// TIA Portal V21 export
FUNCTION_BLOCK "FB301"   // FB301, LAD
TITLE = FB301
{ S7_Optimized_Access := 'TRUE' }
AUTHOR : PRECISE
FAMILY : PRECISE
// FILLING/FINAL VOLUME MAKEUP
// stored: AutoNumber false, MemoryReserve 100, SetENOAutomatically false
   VAR_INPUT
      Enable : Bool;
      Disable : Bool;
      Fault : Bool;
      SecPulse : Bool;
      AlwaysTrue : Bool;
      StartConfirmationPopupSel : Bool;   // StartConfirmationPopupSel: 0-NO/1-YES
      EndConfirmationPopupSel : Bool;   // EndConfirmationPopupSel: 0-NO/1-YES
      FillModeSel : Int;   // Filling Mode Selection: 0-Auto/1-Manual
      FillMethodSel : Int;   // Filling Method Selection: 0-Weight/1-Time
      FillTimeBaseSel : Bool;   // Filling Time Base Selection: 0-second/1-minute
      FillLineSel : Int;   // Filling Line Selection: 0-J tube/1-SBI
      InitialDrainSel : Bool;
      SBIPulsingSel : Bool;
      FinalVolumeMakeupSel : Bool;
      PurgingSel : Bool;
      UtilitySel : Bool;   // Utility Selection: 0-PW/1-WFI
      FillQuantity : Real := 10.0;   // For Filling Method Slection: 0-Weight
      FillTimeMin : Int := 1;   // For Filling Method Slection: 1-Time
      FillTimeSec : Int := 30;   // For Filling Method Slection: 1-Time
      ActualQuantity : Real;   // For Filling Method Slection: 0-Weight
      InflightQuantity : Real;   // For Filling Method Slection: 0-Weight
      ZDVDelay : Int := 3;
      InitialDrainDelay : Int := 10;   // For Initial Drain Selection: Yes
      PurgingTime : Int := 10;   // For Purging Selection: Yes
      SBIOnTime : Int := 3;   // For SBI Pulsing Selection: Yes
      SBIOffTime : Int := 4;   // For SBI Pulsing Selection: Yes
      SetQuantitytoStartPulsing : Real := 10.0;   // For SBI Pulsing Selection: Yes
      FillQuantityTolerance : Real := 3.0;   // For Filling Method Slection: 0-Weight
      PrintInetrval : Int;
   END_VAR
   VAR_OUTPUT
      PWZDV : Bool;   // For Utility Selection: 0-PW
      WFIZDV : Bool;   // For Utility Selection: 1-WFI
      PWLineValves : Bool;   // For Utility Selection: 0-PW
      WFILineValves : Bool;   // For Utility Selection: 1-WFI
      InitialDrainValves : Bool;   // For Initial Drain Selection: Yes
      SBIValve : Bool;   // For Filling Line Selection: 1-SBI
      JTubeValve : Bool;   // For Filling Line Selection: 0-J tube
      AirInletValve : Bool;   // For Purging Selection: Yes
      StartConfirmationPopup : Bool;   // For Start Confirmation Popup Selection: Yes
      EndConfirmationPopup : Bool;   // For End Confirmation Popup Selection: Yes
      ManualPopup : Bool;   // For Filling Mode Selection: 1-Manual
      AlarmFillQuantityExeeded : Bool;
      FillTimeMinPV : DInt;   // For Filling Method Slection: 1-Time
      FillTimeSecPV : DInt;   // For Filling Method Slection: 1-Time
      PrintTrigger : Bool;
      PrintWord : Int;
      PrintStatus : String[50];
   END_VAR
   VAR_IN_OUT
      Start : Bool;
      Stop : Bool;
      Reset : Bool;
      StartConfirmationAck : Bool;   // For Start Confirmation Popup Selection: Yes
      EndConfirmationAck : Bool;   // For End Confirmation Popup Selection: Yes
      ManualAck : Bool;   // For Filling Mode Selection: 1-Manual
      AlarmAck : Bool;
      SpareBtn1 : Bool;
      Running : Bool;
      Selected : Bool;
      Paused : Bool;
      StartConfirmationPopupTemp : Bool;   // For Start Confirmation Popup Selection: Yes
      EndConfirmationPopupTemp : Bool;   // For End Confirmation Popup Selection: Yes
      ManualPopupTemp : Bool;   // For Filling Mode Selection: 1-Manual
      InitialDrainDelayStarted : Bool;
      InitialDrainDelayOver : Bool;
      FillStarted : Bool;
      FillOver : Bool;
      FillOverTemp : Bool;
      InitialDrainDelayPV : Int;
      ActualFillQuantityCalc : Real;   // For Filling Method Slection: 0-Weight
      ActualFillQuantity : Real;   // For Filling Method Slection: 0-Weight
      PulsingStartWeight : Real;   // For SBI Pulsing Selection: Yes
      PurgingTimePV : Int;   // For Purging Selection: Yes
      FillQuantityToleranceCalc : Real := 3.0;   // For Filling Method Slection: 0-Weight
      VesselMaxWeight : Real := 1000.0;
      ResetBatchTimer : Bool;
   END_VAR
   VAR
      ValveOnDelayPV : Int;
      ValveOffDelayPV : Int;
      PrintTriggerTemp : Bool;
      RE1 : Bool;
      RE2 : Bool;
      RE3 : Bool;
      RE4 : Bool;
      RE5 : Bool;
      RE6 : Bool;
      RE7 : Bool;
      FillTimer { S7_SetPoint := 'True'} : "FB101";
      SBIPulsing { S7_SetPoint := 'True'} : "FB102";
      PrintTriggerResetTimer { S7_SetPoint := 'True'} : TON_TIME;
      BtnResetTimer { S7_SetPoint := 'True'} : TON_TIME;
      IEC_Counter_0_Instance { S7_SetPoint := 'True'} : CTU_INT;
   END_VAR
   VAR_TEMP
      STATUS1 : String[40];
      STATUS2 : String[40];
      STATUS3 : String[40];
      STATUS4 : String[40];
      STATUS5 : String[40];
   END_VAR
   VAR_TEMP   // added for the SCL form of the ladder/FBD networks
      _w1 : Bool;
      _w2 : Bool;
      _w3 : Bool;
      _w4 : Bool;
      _w5 : Bool;
      _w6 : Bool;
   END_VAR
BEGIN

REGION Network 1: Running
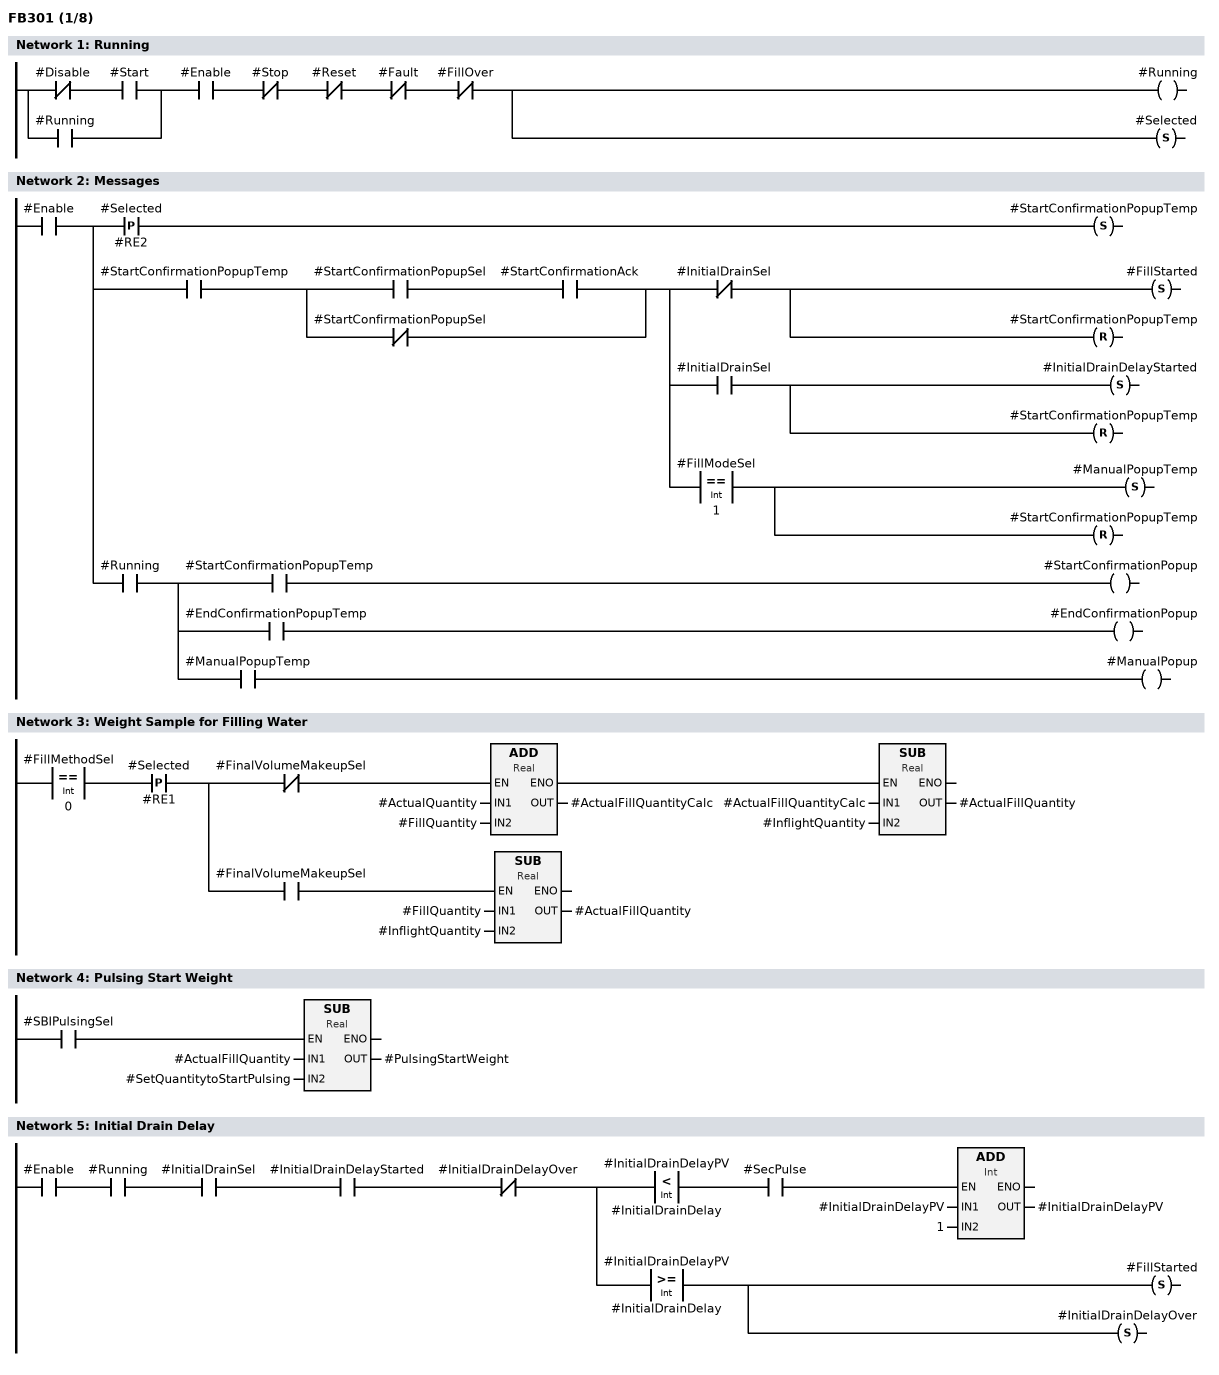
   RUNG wire#powerrail
      I_Contact( #Disable )
      Contact( #Start )
      wire#w1
      Contact( #Enable )
      I_Contact( #Stop )
      I_Contact( #Reset )
      I_Contact( #Fault )
      I_Contact( #FillOver )
      wire#w2
      Coil( #Running )
   END_RUNG
   RUNG wire#powerrail
      Contact( #Running )
   END_RUNG wire#w1
   RUNG wire#w2
      S_Coil( #Selected )
   END_RUNG
   // the same network as SCL:
   #Running := ((NOT #Disable AND #Start) OR #Running) AND #Enable AND NOT #Stop AND NOT #Reset AND NOT #Fault AND NOT #FillOver;
   IF #Running THEN #Selected := TRUE; END_IF;
END_REGION

REGION Network 2: Messages
   RUNG wire#powerrail
      Contact( #Enable )
      wire#w1
      P_Contact(operand := #Selected, bit := #RE2)
      S_Coil( #StartConfirmationPopupTemp )
   END_RUNG
   RUNG wire#w1
      Contact( #StartConfirmationPopupTemp )
      wire#w2
      Contact( #StartConfirmationPopupSel )
      Contact( #StartConfirmationAck )
      wire#w3
      I_Contact( #InitialDrainSel )
      wire#w4
      S_Coil( #FillStarted )
   END_RUNG
   RUNG wire#w2
      I_Contact( #StartConfirmationPopupSel )
   END_RUNG wire#w3
   RUNG wire#w4
      R_Coil( #StartConfirmationPopupTemp )
   END_RUNG
   RUNG wire#w3
      Contact( #InitialDrainSel )
      wire#w5
      S_Coil( #InitialDrainDelayStarted )
   END_RUNG
   RUNG wire#w5
      R_Coil( #StartConfirmationPopupTemp )
   END_RUNG
   RUNG wire#w3
      { S7_Templates := "SrcType := Int" } EQ_Contact(in1 := #FillModeSel, in2 := 1)
      wire#w6
      S_Coil( #ManualPopupTemp )
   END_RUNG
   RUNG wire#w6
      R_Coil( #StartConfirmationPopupTemp )
   END_RUNG
   RUNG wire#w1
      Contact( #Running )
      wire#w7
      Contact( #StartConfirmationPopupTemp )
      Coil( #StartConfirmationPopup )
   END_RUNG
   RUNG wire#w7
      Contact( #EndConfirmationPopupTemp )
      Coil( #EndConfirmationPopup )
   END_RUNG
   RUNG wire#w7
      Contact( #ManualPopupTemp )
      Coil( #ManualPopup )
   END_RUNG
   // the same network as SCL:
   #_w1 := #Enable AND #Selected AND NOT #RE2;   // rising edge of #Selected
   #RE2 := #Selected;
   IF #_w1 THEN #StartConfirmationPopupTemp := TRUE; END_IF;
   #_w2 := #Enable AND #StartConfirmationPopupTemp AND ((#StartConfirmationPopupSel AND #StartConfirmationAck) OR NOT #StartConfirmationPopupSel);
   IF #_w2 AND NOT #InitialDrainSel THEN
       #FillStarted := TRUE;
       #StartConfirmationPopupTemp := FALSE;
   END_IF;
   IF #_w2 AND #InitialDrainSel THEN
       #InitialDrainDelayStarted := TRUE;
       #StartConfirmationPopupTemp := FALSE;
   END_IF;
   IF #_w2 AND (#FillModeSel = 1) THEN
       #ManualPopupTemp := TRUE;
       #StartConfirmationPopupTemp := FALSE;
   END_IF;
   #_w3 := #Enable AND #Running;
   #StartConfirmationPopup := #_w3 AND #StartConfirmationPopupTemp;
   #EndConfirmationPopup := #_w3 AND #EndConfirmationPopupTemp;
   #ManualPopup := #_w3 AND #ManualPopupTemp;
END_REGION

REGION Network 3: Weight Sample for Filling Water
   RUNG wire#powerrail
      { S7_Templates := "SrcType := Int" } EQ_Contact(in1 := #FillMethodSel, in2 := 0)
      P_Contact(operand := #Selected, bit := #RE1)
      wire#w1
      I_Contact( #FinalVolumeMakeupSel )
      { S7_Templates := "SrcType := Real"; S7_GenerateENO := "TRUE" } Add(in1 := #ActualQuantity, in2 := #FillQuantity, out => #ActualFillQuantityCalc)
      { S7_Templates := "SrcType := Real"; S7_GenerateENO := "TRUE" } Sub(in1 := #ActualFillQuantityCalc, in2 := #InflightQuantity, out => #ActualFillQuantity)
   END_RUNG
   RUNG wire#w1
      Contact( #FinalVolumeMakeupSel )
      { S7_Templates := "SrcType := Real"; S7_GenerateENO := "TRUE" } Sub(in1 := #FillQuantity, in2 := #InflightQuantity, out => #ActualFillQuantity)
   END_RUNG
   // the same network as SCL:
   // ENO of a box is taken as its EN; it also drops when the box reports an error
   #_w1 := (#FillMethodSel = 0) AND #Selected AND NOT #RE1;   // rising edge of #Selected
   #RE1 := #Selected;
   IF #_w1 AND NOT #FinalVolumeMakeupSel THEN
       #ActualFillQuantityCalc := #ActualQuantity + #FillQuantity;
       #ActualFillQuantity := #ActualFillQuantityCalc - #InflightQuantity;
   END_IF;
   IF #_w1 AND #FinalVolumeMakeupSel THEN #ActualFillQuantity := #FillQuantity - #InflightQuantity; END_IF;
END_REGION

REGION Network 4: Pulsing Start Weight
   RUNG wire#powerrail
      Contact( #SBIPulsingSel )
      { S7_Templates := "SrcType := Real"; S7_GenerateENO := "TRUE" } Sub(in1 := #ActualFillQuantity, in2 := #SetQuantitytoStartPulsing, out => #PulsingStartWeight)
   END_RUNG
   // the same network as SCL:
   IF #SBIPulsingSel THEN #PulsingStartWeight := #ActualFillQuantity - #SetQuantitytoStartPulsing; END_IF;
END_REGION

REGION Network 5: Initial Drain Delay
   RUNG wire#powerrail
      Contact( #Enable )
      Contact( #Running )
      Contact( #InitialDrainSel )
      Contact( #InitialDrainDelayStarted )
      I_Contact( #InitialDrainDelayOver )
      wire#w1
      { S7_Templates := "SrcType := Int" } LT_Contact(in1 := #InitialDrainDelayPV, in2 := #InitialDrainDelay)
      Contact( #SecPulse )
      { S7_Templates := "SrcType := Int"; S7_GenerateENO := "TRUE" } Add(in1 := #InitialDrainDelayPV, in2 := 1, out => #InitialDrainDelayPV)
   END_RUNG
   RUNG wire#w1
      { S7_Templates := "SrcType := Int" } GE_Contact(in1 := #InitialDrainDelayPV, in2 := #InitialDrainDelay)
      wire#w2
      S_Coil( #FillStarted )
   END_RUNG
   RUNG wire#w2
      S_Coil( #InitialDrainDelayOver )
   END_RUNG
   // the same network as SCL:
   #_w1 := #Enable AND #Running AND #InitialDrainSel AND #InitialDrainDelayStarted AND NOT #InitialDrainDelayOver;
   IF #_w1 AND (#InitialDrainDelayPV < #InitialDrainDelay) AND #SecPulse THEN
       #InitialDrainDelayPV := #InitialDrainDelayPV + 1;
   END_IF;
   IF #_w1 AND (#InitialDrainDelayPV >= #InitialDrainDelay) THEN
       #FillStarted := TRUE;
       #InitialDrainDelayOver := TRUE;
   END_IF;
END_REGION

REGION Network 6: Fill Timer
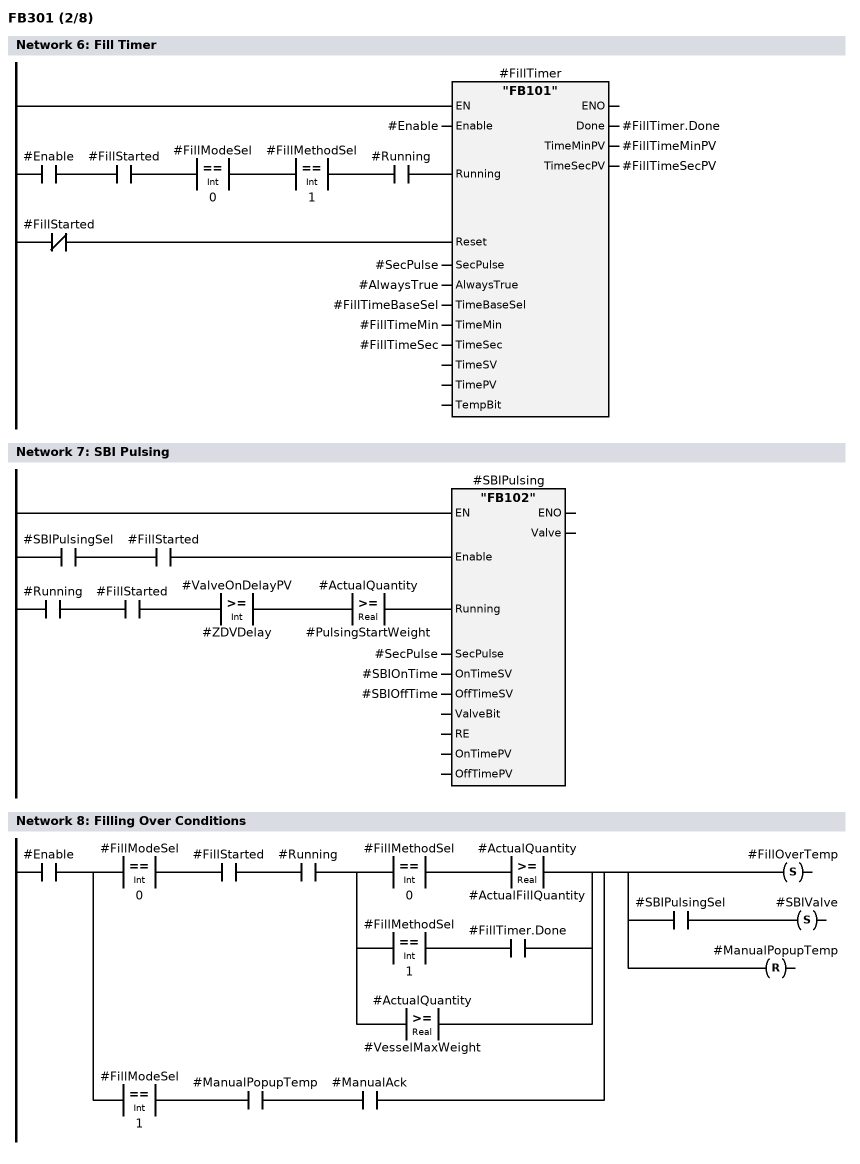
   RUNG wire#powerrail
      #FillTimer(Running := wire#w1, Reset := wire#w2, Enable := #Enable, SecPulse := #SecPulse, AlwaysTrue := #AlwaysTrue, TimeBaseSel := #FillTimeBaseSel, TimeMin := #FillTimeMin, TimeSec := #FillTimeSec, TimeSV :=, TimePV :=, TempBit :=, Done => #FillTimer.Done, TimeMinPV => #FillTimeMinPV, TimeSecPV => #FillTimeSecPV)
   END_RUNG
   RUNG wire#powerrail
      Contact( #Enable )
      Contact( #FillStarted )
      { S7_Templates := "SrcType := Int" } EQ_Contact(in1 := #FillModeSel, in2 := 0)
      { S7_Templates := "SrcType := Int" } EQ_Contact(in1 := #FillMethodSel, in2 := 1)
      Contact( #Running )
   END_RUNG wire#w1
   RUNG wire#powerrail
      I_Contact( #FillStarted )
   END_RUNG wire#w2
   // the same network as SCL:
   #FillTimer(Enable := #Enable,   // "FB101"
              Running := #Enable AND #FillStarted AND (#FillModeSel = 0) AND (#FillMethodSel = 1) AND #Running,
              Reset := NOT #FillStarted,
              SecPulse := #SecPulse,
              AlwaysTrue := #AlwaysTrue,
              TimeBaseSel := #FillTimeBaseSel,
              TimeMin := #FillTimeMin,
              TimeSec := #FillTimeSec,
              Done => #FillTimer.Done,
              TimeMinPV => #FillTimeMinPV,
              TimeSecPV => #FillTimeSecPV);
END_REGION

REGION Network 7: SBI Pulsing
   RUNG wire#powerrail
      #SBIPulsing(Enable := wire#w1, Running := wire#w2, SecPulse := #SecPulse, OnTimeSV := #SBIOnTime, OffTimeSV := #SBIOffTime, ValveBit :=, RE :=, OnTimePV :=, OffTimePV :=, Valve =>)
   END_RUNG
   RUNG wire#powerrail
      Contact( #SBIPulsingSel )
      Contact( #FillStarted )
   END_RUNG wire#w1
   RUNG wire#powerrail
      Contact( #Running )
      Contact( #FillStarted )
      { S7_Templates := "SrcType := Int" } GE_Contact(in1 := #ValveOnDelayPV, in2 := #ZDVDelay)
      { S7_Templates := "SrcType := Real" } GE_Contact(in1 := #ActualQuantity, in2 := #PulsingStartWeight)
   END_RUNG wire#w2
   // the same network as SCL:
   #SBIPulsing(Enable := #SBIPulsingSel AND #FillStarted,   // "FB102"
               Running := #Running AND #FillStarted AND (#ValveOnDelayPV >= #ZDVDelay) AND (#ActualQuantity >= #PulsingStartWeight),
               SecPulse := #SecPulse,
               OnTimeSV := #SBIOnTime,
               OffTimeSV := #SBIOffTime);
END_REGION

REGION Network 8: Filling Over Conditions
   RUNG wire#powerrail
      Contact( #Enable )
      wire#w1
      { S7_Templates := "SrcType := Int" } EQ_Contact(in1 := #FillModeSel, in2 := 0)
      Contact( #FillStarted )
      Contact( #Running )
      wire#w2
      { S7_Templates := "SrcType := Int" } EQ_Contact(in1 := #FillMethodSel, in2 := 0)
      { S7_Templates := "SrcType := Real" } GE_Contact(in1 := #ActualQuantity, in2 := #ActualFillQuantity)
      wire#w3
      S_Coil( #FillOverTemp )
   END_RUNG
   RUNG wire#w2
      { S7_Templates := "SrcType := Int" } EQ_Contact(in1 := #FillMethodSel, in2 := 1)
      Contact( #FillTimer.Done )
   END_RUNG wire#w3
   RUNG wire#w2
      { S7_Templates := "SrcType := Real" } GE_Contact(in1 := #ActualQuantity, in2 := #VesselMaxWeight)
   END_RUNG wire#w3
   RUNG wire#w1
      { S7_Templates := "SrcType := Int" } EQ_Contact(in1 := #FillModeSel, in2 := 1)
      Contact( #ManualPopupTemp )
      Contact( #ManualAck )
   END_RUNG wire#w3
   RUNG wire#w3
      Contact( #SBIPulsingSel )
      S_Coil( #SBIValve )
   END_RUNG
   RUNG wire#w3
      R_Coil( #ManualPopupTemp )
   END_RUNG
   // the same network as SCL:
   #_w1 := #Enable AND (((#FillModeSel = 0) AND #FillStarted AND #Running AND (((#FillMethodSel = 0) AND (#ActualQuantity >= #ActualFillQuantity)) OR ((#FillMethodSel = 1) AND #FillTimer.Done) OR (#ActualQuantity >= #VesselMaxWeight))) OR ((#FillModeSel = 1) AND #ManualPopupTemp AND #ManualAck));
   IF #_w1 THEN #FillOverTemp := TRUE; END_IF;
   IF #_w1 AND #SBIPulsingSel THEN #SBIValve := TRUE; END_IF;
   IF #_w1 THEN #ManualPopupTemp := FALSE; END_IF;
END_REGION

REGION Network 9: Purging Timer
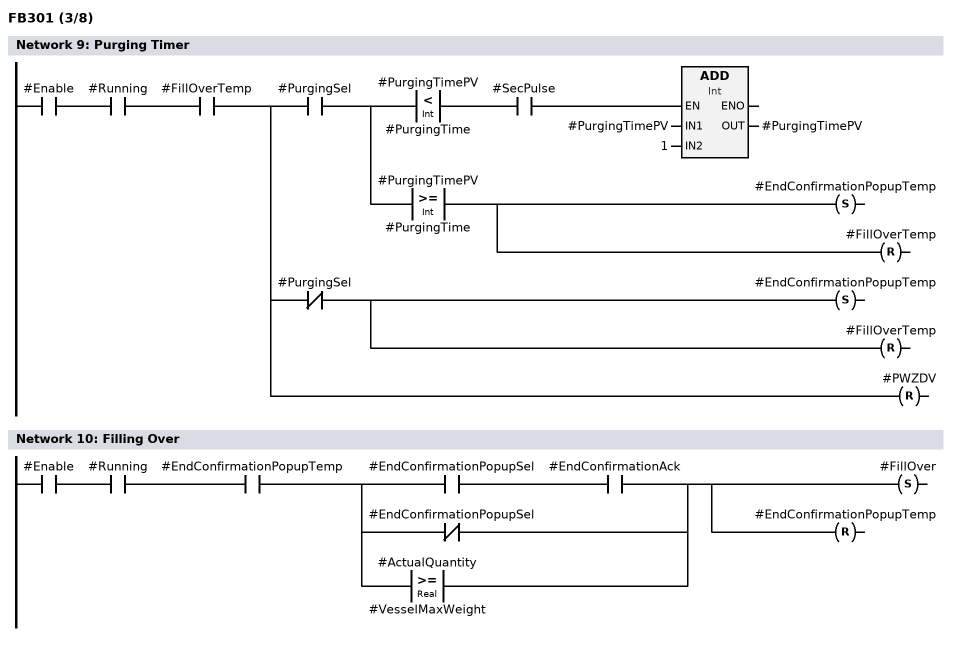
   RUNG wire#powerrail
      Contact( #Enable )
      Contact( #Running )
      Contact( #FillOverTemp )
      wire#w1
      Contact( #PurgingSel )
      wire#w2
      { S7_Templates := "SrcType := Int" } LT_Contact(in1 := #PurgingTimePV, in2 := #PurgingTime)
      Contact( #SecPulse )
      { S7_Templates := "SrcType := Int"; S7_GenerateENO := "TRUE" } Add(in1 := #PurgingTimePV, in2 := 1, out => #PurgingTimePV)
   END_RUNG
   RUNG wire#w2
      { S7_Templates := "SrcType := Int" } GE_Contact(in1 := #PurgingTimePV, in2 := #PurgingTime)
      wire#w3
      S_Coil( #EndConfirmationPopupTemp )
   END_RUNG
   RUNG wire#w3
      R_Coil( #FillOverTemp )
   END_RUNG
   RUNG wire#w1
      I_Contact( #PurgingSel )
      wire#w4
      S_Coil( #EndConfirmationPopupTemp )
   END_RUNG
   RUNG wire#w4
      R_Coil( #FillOverTemp )
   END_RUNG
   RUNG wire#w1
      R_Coil( #PWZDV )
   END_RUNG
   // the same network as SCL:
   #_w1 := #Enable AND #Running AND #FillOverTemp;
   #_w2 := #_w1 AND #PurgingSel;
   IF #_w2 AND (#PurgingTimePV < #PurgingTime) AND #SecPulse THEN
       #PurgingTimePV := #PurgingTimePV + 1;
   END_IF;
   IF #_w2 AND (#PurgingTimePV >= #PurgingTime) THEN
       #EndConfirmationPopupTemp := TRUE;
       #FillOverTemp := FALSE;
   END_IF;
   IF #_w1 AND NOT #PurgingSel THEN
       #EndConfirmationPopupTemp := TRUE;
       #FillOverTemp := FALSE;
   END_IF;
   IF #_w1 THEN #PWZDV := FALSE; END_IF;
END_REGION

REGION Network 10: Filling Over
   RUNG wire#powerrail
      Contact( #Enable )
      Contact( #Running )
      Contact( #EndConfirmationPopupTemp )
      wire#w1
      Contact( #EndConfirmationPopupSel )
      Contact( #EndConfirmationAck )
      wire#w2
      S_Coil( #FillOver )
   END_RUNG
   RUNG wire#w1
      I_Contact( #EndConfirmationPopupSel )
   END_RUNG wire#w2
   RUNG wire#w1
      { S7_Templates := "SrcType := Real" } GE_Contact(in1 := #ActualQuantity, in2 := #VesselMaxWeight)
   END_RUNG wire#w2
   RUNG wire#w2
      R_Coil( #EndConfirmationPopupTemp )
   END_RUNG
   // the same network as SCL:
   IF #Enable AND #Running AND #EndConfirmationPopupTemp AND ((#EndConfirmationPopupSel AND #EndConfirmationAck) OR NOT #EndConfirmationPopupSel OR (#ActualQuantity >= #VesselMaxWeight)) THEN
       #FillOver := TRUE;
       #EndConfirmationPopupTemp := FALSE;
   END_IF;
END_REGION

REGION Network 11: Output On
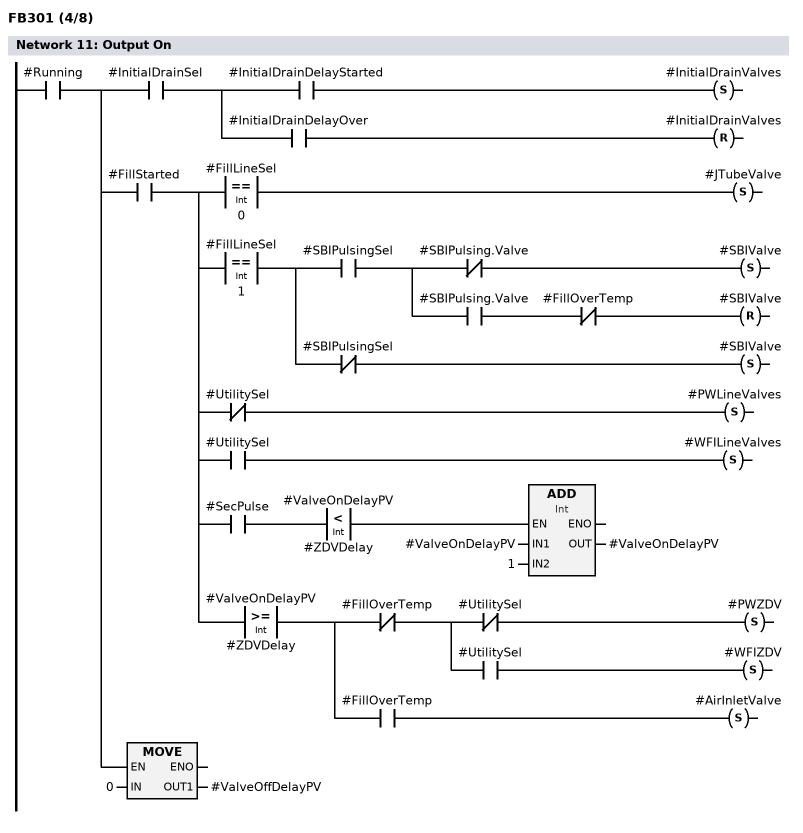
   RUNG wire#powerrail
      Contact( #Running )
      wire#w1
      Contact( #InitialDrainSel )
      wire#w2
      Contact( #InitialDrainDelayStarted )
      S_Coil( #InitialDrainValves )
   END_RUNG
   RUNG wire#w2
      Contact( #InitialDrainDelayOver )
      R_Coil( #InitialDrainValves )
   END_RUNG
   RUNG wire#w1
      Contact( #FillStarted )
      wire#w3
      { S7_Templates := "SrcType := Int" } EQ_Contact(in1 := #FillLineSel, in2 := 0)
      S_Coil( #JTubeValve )
   END_RUNG
   RUNG wire#w3
      { S7_Templates := "SrcType := Int" } EQ_Contact(in1 := #FillLineSel, in2 := 1)
      wire#w4
      Contact( #SBIPulsingSel )
      wire#w5
      I_Contact( #SBIPulsing.Valve )
      S_Coil( #SBIValve )
   END_RUNG
   RUNG wire#w5
      Contact( #SBIPulsing.Valve )
      I_Contact( #FillOverTemp )
      R_Coil( #SBIValve )
   END_RUNG
   RUNG wire#w4
      I_Contact( #SBIPulsingSel )
      S_Coil( #SBIValve )
   END_RUNG
   RUNG wire#w3
      I_Contact( #UtilitySel )
      S_Coil( #PWLineValves )
   END_RUNG
   RUNG wire#w3
      Contact( #UtilitySel )
      S_Coil( #WFILineValves )
   END_RUNG
   RUNG wire#w3
      Contact( #SecPulse )
      { S7_Templates := "SrcType := Int" } LT_Contact(in1 := #ValveOnDelayPV, in2 := #ZDVDelay)
      { S7_Templates := "SrcType := Int"; S7_GenerateENO := "TRUE" } Add(in1 := #ValveOnDelayPV, in2 := 1, out => #ValveOnDelayPV)
   END_RUNG
   RUNG wire#w3
      { S7_Templates := "SrcType := Int" } GE_Contact(in1 := #ValveOnDelayPV, in2 := #ZDVDelay)
      wire#w6
      I_Contact( #FillOverTemp )
      wire#w7
      I_Contact( #UtilitySel )
      S_Coil( #PWZDV )
   END_RUNG
   RUNG wire#w7
      Contact( #UtilitySel )
      S_Coil( #WFIZDV )
   END_RUNG
   RUNG wire#w6
      Contact( #FillOverTemp )
      S_Coil( #AirInletValve )
   END_RUNG
   RUNG wire#w1
      { S7_GenerateENO := "TRUE" } Move(in := 0, out1 => #ValveOffDelayPV)
   END_RUNG
   // the same network as SCL:
   #_w1 := #Running AND #InitialDrainSel;
   IF #_w1 AND #InitialDrainDelayStarted THEN #InitialDrainValves := TRUE; END_IF;
   IF #_w1 AND #InitialDrainDelayOver THEN #InitialDrainValves := FALSE; END_IF;
   #_w2 := #Running AND #FillStarted;
   IF #_w2 AND (#FillLineSel = 0) THEN #JTubeValve := TRUE; END_IF;
   #_w3 := #_w2 AND (#FillLineSel = 1);
   #_w4 := #_w3 AND #SBIPulsingSel;
   IF #_w4 AND NOT #SBIPulsing.Valve THEN #SBIValve := TRUE; END_IF;
   IF #_w4 AND #SBIPulsing.Valve AND NOT #FillOverTemp THEN #SBIValve := FALSE; END_IF;
   IF #_w3 AND NOT #SBIPulsingSel THEN #SBIValve := TRUE; END_IF;
   IF #_w2 AND NOT #UtilitySel THEN #PWLineValves := TRUE; END_IF;
   IF #_w2 AND #UtilitySel THEN #WFILineValves := TRUE; END_IF;
   IF #_w2 AND #SecPulse AND (#ValveOnDelayPV < #ZDVDelay) THEN
       #ValveOnDelayPV := #ValveOnDelayPV + 1;
   END_IF;
   #_w5 := #_w2 AND (#ValveOnDelayPV >= #ZDVDelay);
   #_w6 := #_w5 AND NOT #FillOverTemp;
   IF #_w6 AND NOT #UtilitySel THEN #PWZDV := TRUE; END_IF;
   IF #_w6 AND #UtilitySel THEN #WFIZDV := TRUE; END_IF;
   IF #_w5 AND #FillOverTemp THEN #AirInletValve := TRUE; END_IF;
   IF #Running THEN #ValveOffDelayPV := 0; END_IF;
END_REGION

REGION Network 12: Output Off
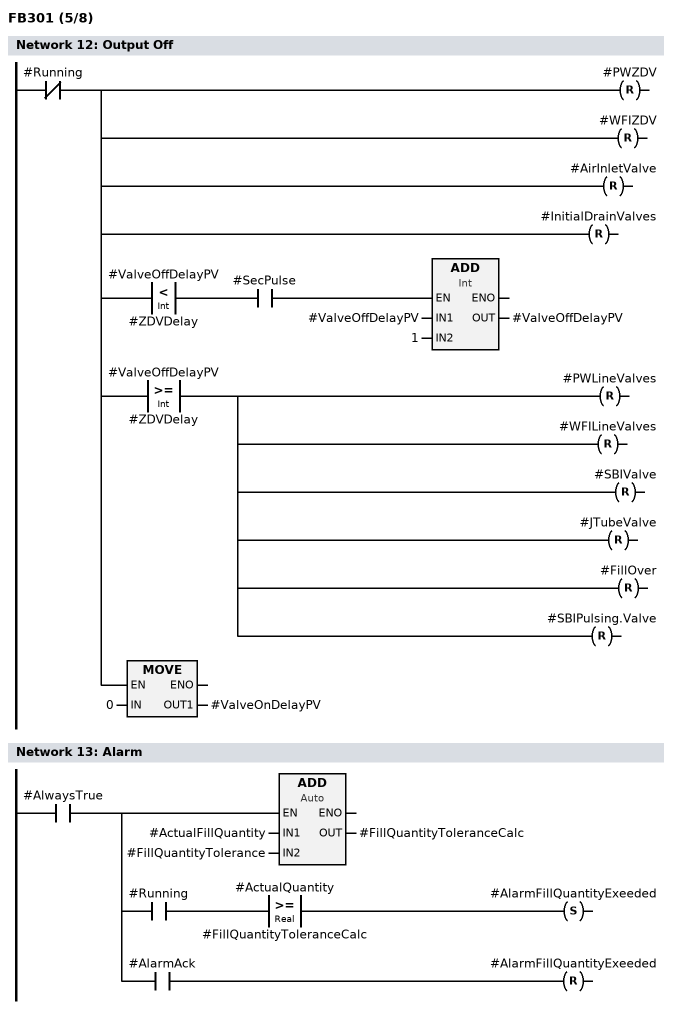
   RUNG wire#powerrail
      I_Contact( #Running )
      wire#w1
      R_Coil( #PWZDV )
   END_RUNG
   RUNG wire#w1
      R_Coil( #WFIZDV )
   END_RUNG
   RUNG wire#w1
      R_Coil( #AirInletValve )
   END_RUNG
   RUNG wire#w1
      R_Coil( #InitialDrainValves )
   END_RUNG
   RUNG wire#w1
      { S7_Templates := "SrcType := Int" } LT_Contact(in1 := #ValveOffDelayPV, in2 := #ZDVDelay)
      Contact( #SecPulse )
      { S7_Templates := "SrcType := Int"; S7_GenerateENO := "TRUE" } Add(in1 := #ValveOffDelayPV, in2 := 1, out => #ValveOffDelayPV)
   END_RUNG
   RUNG wire#w1
      { S7_Templates := "SrcType := Int" } GE_Contact(in1 := #ValveOffDelayPV, in2 := #ZDVDelay)
      wire#w2
      R_Coil( #PWLineValves )
   END_RUNG
   RUNG wire#w2
      R_Coil( #WFILineValves )
   END_RUNG
   RUNG wire#w2
      R_Coil( #SBIValve )
   END_RUNG
   RUNG wire#w2
      R_Coil( #JTubeValve )
   END_RUNG
   RUNG wire#w2
      R_Coil( #FillOver )
   END_RUNG
   RUNG wire#w2
      R_Coil( #SBIPulsing.Valve )
   END_RUNG
   RUNG wire#w1
      { S7_GenerateENO := "TRUE" } Move(in := 0, out1 => #ValveOnDelayPV)
   END_RUNG
   // the same network as SCL:
   IF NOT #Running THEN
       #PWZDV := FALSE;
       #WFIZDV := FALSE;
       #AirInletValve := FALSE;
       #InitialDrainValves := FALSE;
   END_IF;
   IF NOT #Running AND (#ValveOffDelayPV < #ZDVDelay) AND #SecPulse THEN
       #ValveOffDelayPV := #ValveOffDelayPV + 1;
   END_IF;
   IF NOT #Running AND (#ValveOffDelayPV >= #ZDVDelay) THEN
       #PWLineValves := FALSE;
       #WFILineValves := FALSE;
       #SBIValve := FALSE;
       #JTubeValve := FALSE;
       #FillOver := FALSE;
       #SBIPulsing.Valve := FALSE;
   END_IF;
   IF NOT #Running THEN #ValveOnDelayPV := 0; END_IF;
END_REGION

REGION Network 13: Alarm
   RUNG wire#powerrail
      Contact( #AlwaysTrue )
      wire#w1
      Add(in1 := #ActualFillQuantity, in2 := #FillQuantityTolerance, out => #FillQuantityToleranceCalc)
   END_RUNG
   RUNG wire#w1
      Contact( #Running )
      { S7_Templates := "SrcType := Real" } GE_Contact(in1 := #ActualQuantity, in2 := #FillQuantityToleranceCalc)
      S_Coil( #AlarmFillQuantityExeeded )
   END_RUNG
   RUNG wire#w1
      Contact( #AlarmAck )
      R_Coil( #AlarmFillQuantityExeeded )
   END_RUNG
   // the same network as SCL:
   IF #AlwaysTrue THEN #FillQuantityToleranceCalc := #ActualFillQuantity + #FillQuantityTolerance; END_IF;
   IF #AlwaysTrue AND #Running AND (#ActualQuantity >= #FillQuantityToleranceCalc) THEN
       #AlarmFillQuantityExeeded := TRUE;
   END_IF;
   IF #AlwaysTrue AND #AlarmAck THEN #AlarmFillQuantityExeeded := FALSE; END_IF;
END_REGION

REGION Network 14: Event Status
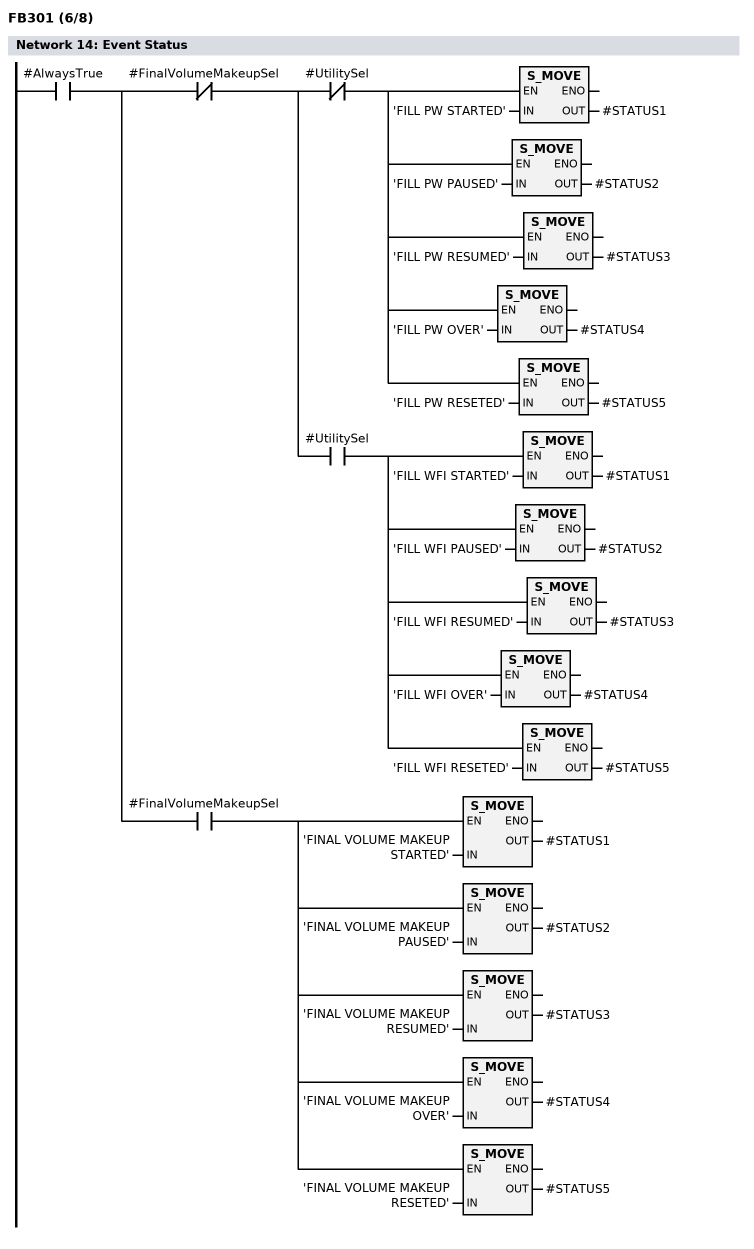
   RUNG wire#powerrail
      Contact( #AlwaysTrue )
      wire#w1
      I_Contact( #FinalVolumeMakeupSel )
      wire#w2
      I_Contact( #UtilitySel )
      wire#w3
      S_Move(in := 'FILL PW STARTED', out => #STATUS1)
   END_RUNG
   RUNG wire#w3
      S_Move(in := 'FILL PW PAUSED', out => #STATUS2)
   END_RUNG
   RUNG wire#w3
      S_Move(in := 'FILL PW RESUMED', out => #STATUS3)
   END_RUNG
   RUNG wire#w3
      S_Move(in := 'FILL PW OVER', out => #STATUS4)
   END_RUNG
   RUNG wire#w3
      S_Move(in := 'FILL PW RESETED', out => #STATUS5)
   END_RUNG
   RUNG wire#w2
      Contact( #UtilitySel )
      wire#w4
      S_Move(in := 'FILL WFI STARTED', out => #STATUS1)
   END_RUNG
   RUNG wire#w4
      S_Move(in := 'FILL WFI PAUSED', out => #STATUS2)
   END_RUNG
   RUNG wire#w4
      S_Move(in := 'FILL WFI RESUMED', out => #STATUS3)
   END_RUNG
   RUNG wire#w4
      S_Move(in := 'FILL WFI OVER', out => #STATUS4)
   END_RUNG
   RUNG wire#w4
      S_Move(in := 'FILL WFI RESETED', out => #STATUS5)
   END_RUNG
   RUNG wire#w1
      Contact( #FinalVolumeMakeupSel )
      wire#w5
      S_Move(in := 'FINAL VOLUME MAKEUP STARTED', out => #STATUS1)
   END_RUNG
   RUNG wire#w5
      S_Move(in := 'FINAL VOLUME MAKEUP PAUSED', out => #STATUS2)
   END_RUNG
   RUNG wire#w5
      S_Move(in := 'FINAL VOLUME MAKEUP RESUMED', out => #STATUS3)
   END_RUNG
   RUNG wire#w5
      S_Move(in := 'FINAL VOLUME MAKEUP OVER', out => #STATUS4)
   END_RUNG
   RUNG wire#w5
      S_Move(in := 'FINAL VOLUME MAKEUP RESETED', out => #STATUS5)
   END_RUNG
   // the same network as SCL:
   #_w1 := #AlwaysTrue AND NOT #FinalVolumeMakeupSel;
   IF #_w1 AND NOT #UtilitySel THEN
       #STATUS1 := 'FILL PW STARTED';
       #STATUS2 := 'FILL PW PAUSED';
       #STATUS3 := 'FILL PW RESUMED';
       #STATUS4 := 'FILL PW OVER';
       #STATUS5 := 'FILL PW RESETED';
   END_IF;
   IF #_w1 AND #UtilitySel THEN
       #STATUS1 := 'FILL WFI STARTED';
       #STATUS2 := 'FILL WFI PAUSED';
       #STATUS3 := 'FILL WFI RESUMED';
       #STATUS4 := 'FILL WFI OVER';
       #STATUS5 := 'FILL WFI RESETED';
   END_IF;
   IF #AlwaysTrue AND #FinalVolumeMakeupSel THEN
       #STATUS1 := 'FINAL VOLUME MAKEUP STARTED';
       #STATUS2 := 'FINAL VOLUME MAKEUP PAUSED';
       #STATUS3 := 'FINAL VOLUME MAKEUP RESUMED';
       #STATUS4 := 'FINAL VOLUME MAKEUP OVER';
       #STATUS5 := 'FINAL VOLUME MAKEUP RESETED';
   END_IF;
END_REGION

REGION Network 15: Print Logic
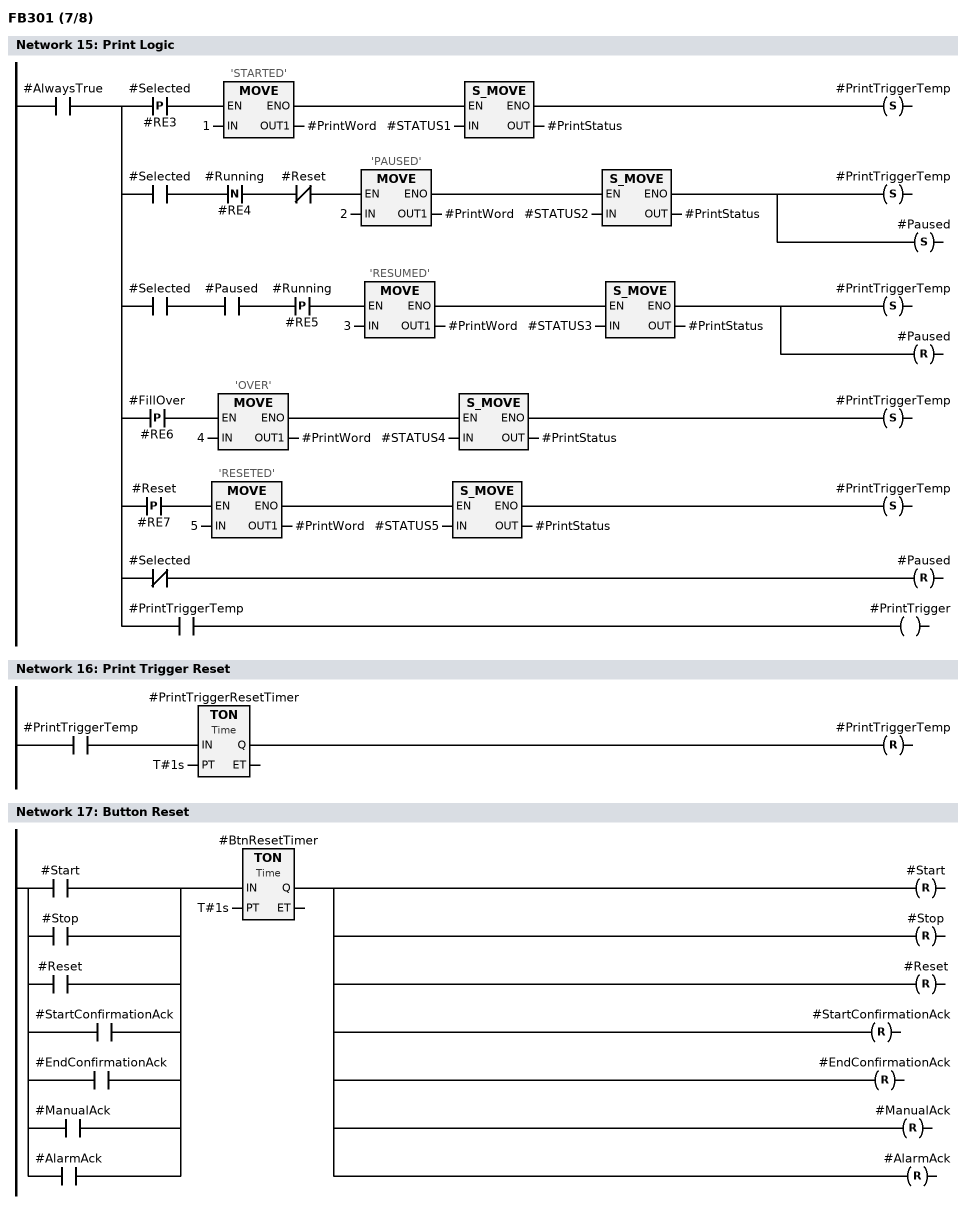
   RUNG wire#powerrail
      Contact( #AlwaysTrue )
      wire#w1
      P_Contact(operand := #Selected, bit := #RE3)
      { S7_GenerateENO := "TRUE" } Move(in := 1, out1 => #PrintWord)   // 'STARTED'
      S_Move(in := #STATUS1, out => #PrintStatus)
      S_Coil( #PrintTriggerTemp )
   END_RUNG
   RUNG wire#w1
      Contact( #Selected )
      N_Contact(operand := #Running, bit := #RE4)
      I_Contact( #Reset )
      { S7_GenerateENO := "TRUE" } Move(in := 2, out1 => #PrintWord)   // 'PAUSED'
      S_Move(in := #STATUS2, out => #PrintStatus)
      wire#w2
      S_Coil( #PrintTriggerTemp )
   END_RUNG
   RUNG wire#w2
      S_Coil( #Paused )
   END_RUNG
   RUNG wire#w1
      Contact( #Selected )
      Contact( #Paused )
      P_Contact(operand := #Running, bit := #RE5)
      { S7_GenerateENO := "TRUE" } Move(in := 3, out1 => #PrintWord)   // 'RESUMED'
      S_Move(in := #STATUS3, out => #PrintStatus)
      wire#w3
      S_Coil( #PrintTriggerTemp )
   END_RUNG
   RUNG wire#w3
      R_Coil( #Paused )
   END_RUNG
   RUNG wire#w1
      P_Contact(operand := #FillOver, bit := #RE6)
      { S7_GenerateENO := "TRUE" } Move(in := 4, out1 => #PrintWord)   // 'OVER'
      S_Move(in := #STATUS4, out => #PrintStatus)
      S_Coil( #PrintTriggerTemp )
   END_RUNG
   RUNG wire#w1
      P_Contact(operand := #Reset, bit := #RE7)
      { S7_GenerateENO := "TRUE" } Move(in := 5, out1 => #PrintWord)   // 'RESETED'
      S_Move(in := #STATUS5, out => #PrintStatus)
      S_Coil( #PrintTriggerTemp )
   END_RUNG
   RUNG wire#w1
      I_Contact( #Selected )
      R_Coil( #Paused )
   END_RUNG
   RUNG wire#w1
      Contact( #PrintTriggerTemp )
      Coil( #PrintTrigger )
   END_RUNG
   // the same network as SCL:
   // ENO of a box is taken as its EN; it also drops when the box reports an error
   #_w1 := #AlwaysTrue AND #Selected AND NOT #RE3;   // rising edge of #Selected
   #RE3 := #Selected;
   IF #_w1 THEN
       #PrintWord := 1;   // 'STARTED'
       #PrintStatus := #STATUS1;
       #PrintTriggerTemp := TRUE;
   END_IF;
   #_w2 := #AlwaysTrue AND #Selected AND NOT #Running AND #RE4;   // falling edge of #Running
   #RE4 := #Running;
   IF #_w2 AND NOT #Reset THEN
       #PrintWord := 2;   // 'PAUSED'
       #PrintStatus := #STATUS2;
       #PrintTriggerTemp := TRUE;
       #Paused := TRUE;
   END_IF;
   #_w3 := #AlwaysTrue AND #Selected AND #Paused AND #Running AND NOT #RE5;   // rising edge of #Running
   #RE5 := #Running;
   IF #_w3 THEN
       #PrintWord := 3;   // 'RESUMED'
       #PrintStatus := #STATUS3;
       #PrintTriggerTemp := TRUE;
       #Paused := FALSE;
   END_IF;
   #_w4 := #AlwaysTrue AND #FillOver AND NOT #RE6;   // rising edge of #FillOver
   #RE6 := #FillOver;
   IF #_w4 THEN
       #PrintWord := 4;   // 'OVER'
       #PrintStatus := #STATUS4;
       #PrintTriggerTemp := TRUE;
   END_IF;
   #_w5 := #AlwaysTrue AND #Reset AND NOT #RE7;   // rising edge of #Reset
   #RE7 := #Reset;
   IF #_w5 THEN
       #PrintWord := 5;   // 'RESETED'
       #PrintStatus := #STATUS5;
       #PrintTriggerTemp := TRUE;
   END_IF;
   IF #AlwaysTrue AND NOT #Selected THEN #Paused := FALSE; END_IF;
   #PrintTrigger := #AlwaysTrue AND #PrintTriggerTemp;
END_REGION

REGION Network 16: Print Trigger Reset
   RUNG wire#powerrail
      Contact( #PrintTriggerTemp )
      { S7_Templates := "time_type := Time" } #PrintTriggerResetTimer.TON(pt := T#1s, et =>)
      R_Coil( #PrintTriggerTemp )
   END_RUNG
   // the same network as SCL:
   #PrintTriggerResetTimer(IN := #PrintTriggerTemp, PT := T#1s);   // TON
   IF #PrintTriggerResetTimer.Q THEN #PrintTriggerTemp := FALSE; END_IF;
END_REGION

REGION Network 17: Button Reset
   RUNG wire#powerrail
      Contact( #Start )
      wire#w1
      { S7_Templates := "time_type := Time" } #BtnResetTimer.TON(pt := T#1s, et =>)
      wire#w2
      R_Coil( #Start )
   END_RUNG
   RUNG wire#powerrail
      Contact( #Stop )
   END_RUNG wire#w1
   RUNG wire#powerrail
      Contact( #Reset )
   END_RUNG wire#w1
   RUNG wire#powerrail
      Contact( #StartConfirmationAck )
   END_RUNG wire#w1
   RUNG wire#powerrail
      Contact( #EndConfirmationAck )
   END_RUNG wire#w1
   RUNG wire#powerrail
      Contact( #ManualAck )
   END_RUNG wire#w1
   RUNG wire#powerrail
      Contact( #AlarmAck )
   END_RUNG wire#w1
   RUNG wire#w2
      R_Coil( #Stop )
   END_RUNG
   RUNG wire#w2
      R_Coil( #Reset )
   END_RUNG
   RUNG wire#w2
      R_Coil( #StartConfirmationAck )
   END_RUNG
   RUNG wire#w2
      R_Coil( #EndConfirmationAck )
   END_RUNG
   RUNG wire#w2
      R_Coil( #ManualAck )
   END_RUNG
   RUNG wire#w2
      R_Coil( #AlarmAck )
   END_RUNG
   // the same network as SCL:
   #BtnResetTimer(IN := #Start OR #Stop OR #Reset OR #StartConfirmationAck OR #EndConfirmationAck OR #ManualAck OR #AlarmAck,   // TON
                  PT := T#1s);
   IF #BtnResetTimer.Q THEN
       #Start := FALSE;
       #Stop := FALSE;
       #Reset := FALSE;
       #StartConfirmationAck := FALSE;
       #EndConfirmationAck := FALSE;
       #ManualAck := FALSE;
       #AlarmAck := FALSE;
   END_IF;
END_REGION

REGION Network 18: Reset
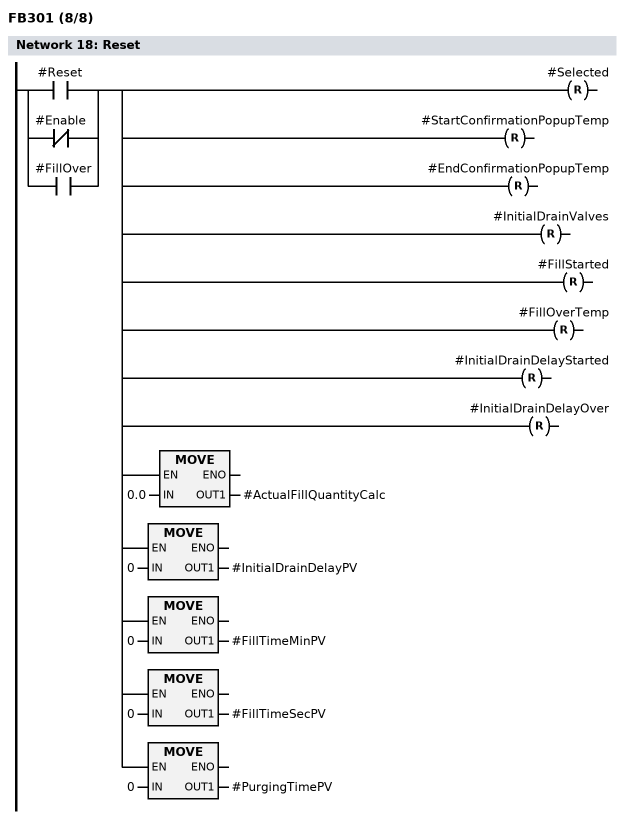
   RUNG wire#powerrail
      Contact( #Reset )
      wire#w1
      R_Coil( #Selected )
   END_RUNG
   RUNG wire#powerrail
      I_Contact( #Enable )
   END_RUNG wire#w1
   RUNG wire#powerrail
      Contact( #FillOver )
   END_RUNG wire#w1
   RUNG wire#w1
      R_Coil( #StartConfirmationPopupTemp )
   END_RUNG
   RUNG wire#w1
      R_Coil( #EndConfirmationPopupTemp )
   END_RUNG
   RUNG wire#w1
      R_Coil( #InitialDrainValves )
   END_RUNG
   RUNG wire#w1
      R_Coil( #FillStarted )
   END_RUNG
   RUNG wire#w1
      R_Coil( #FillOverTemp )
   END_RUNG
   RUNG wire#w1
      R_Coil( #InitialDrainDelayStarted )
   END_RUNG
   RUNG wire#w1
      R_Coil( #InitialDrainDelayOver )
   END_RUNG
   RUNG wire#w1
      { S7_GenerateENO := "TRUE" } Move(in := 0.0, out1 => #ActualFillQuantityCalc)
   END_RUNG
   RUNG wire#w1
      { S7_GenerateENO := "TRUE" } Move(in := 0, out1 => #InitialDrainDelayPV)
   END_RUNG
   RUNG wire#w1
      { S7_GenerateENO := "TRUE" } Move(in := 0, out1 => #FillTimeMinPV)
   END_RUNG
   RUNG wire#w1
      { S7_GenerateENO := "TRUE" } Move(in := 0, out1 => #FillTimeSecPV)
   END_RUNG
   RUNG wire#w1
      { S7_GenerateENO := "TRUE" } Move(in := 0, out1 => #PurgingTimePV)
   END_RUNG
   // the same network as SCL:
   IF #Reset OR NOT #Enable OR #FillOver THEN
       #Selected := FALSE;
       #StartConfirmationPopupTemp := FALSE;
       #EndConfirmationPopupTemp := FALSE;
       #InitialDrainValves := FALSE;
       #FillStarted := FALSE;
       #FillOverTemp := FALSE;
       #InitialDrainDelayStarted := FALSE;
       #InitialDrainDelayOver := FALSE;
       #ActualFillQuantityCalc := 0.0;
       #InitialDrainDelayPV := 0;
       #FillTimeMinPV := 0;
       #FillTimeSecPV := 0;
       #PurgingTimePV := 0;
   END_IF;
END_REGION
END_FUNCTION_BLOCK
